(* Logix 5000 project; controller test vendor 1 type 14 code 151 rev 32.13; software revision 32.02; part 4 of 4 *)
(* tags used below, declared in another part *)
   _i : DINT;
   _J : INT;
   _n : DINT;
   _T : DINT;
   _z : DINT;
   AirDown : CAM_PROFILE[1010];
   AirUp : CAM_PROFILE[1010];
   avgCrsDyn : REAL;   // 1 min avg of dynamic respiratory system compliance in ml/cmH2O, from measAvgCalc()
   avgCrsQStat : REAL;   // 1 min avg of quasistatic respiratory system compliance in ml/cmH2O, from measAvgCalc()
   avgFlowImax : REAL;   // 1 min avg of max insp flow in l/min, from measAvgCalc()
   avgMV : REAL;   // 1 min avg of minute ventilation in l/min, from measAvgCalc()
   avgPEEP : REAL;   // 1 min avg of positive end expiratory pressure in cmH2O, from measAvgCalc()
   avgPpeak : REAL;   // 1 min avg of peak insp pressure in cmH2O, from measAvgCalc()
   avgPplat : REAL;   // 1 min avg of plateau insp pressure in cmH2O, from measAvgCalc()
   avgRaw : REAL;   // 1 min avg of airway resistance in cmH2O/l/s, from measAvgCalc()
   avgRR : REAL;   // 1 min avg of respiratory rate in 1/min, from measAvgCalc()
   avgVti : REAL;   // 1 min avg of insp tidal volume in ml, from measAvgCalc()
   BackingTag : MOTION_INSTRUCTION;
   BreathDuration : INT;
   BreathDurationArr : REAL[50];   // 50 length array with seconds for each breath for calculation of minute avgVentStateArr. Calcualted from knowing meas at
   CalcNewData : BOOL;
   CrsDyn : REAL;   // dynamic respiraotry system compliance in ml/cmH2O
   CrsDynArr : REAL[50];   // 50 length array with dynamic respiraotry system compliance in ml/cmH2O, from measCalc()
   CrsQStat : REAL;   // quasistatic respiratory system compliance in ml/cmH2O
   CrsQStatArr : REAL[50];   // 50 length array with quasistatic respiratory system compliance in ml/cmH2O, from measCalc()
   DymmyMaster : AXIS_VIRTUAL;
   DymmySlave : AXIS_VIRTUAL;
   endI : DINT;
   EndPoint : INT;
   Exp : BOOL;
   expEndI : INT;
   expStartI : INT;
   FillLoop : AOI_FillArray_Real2D;
   FlowArrMem : REAL[1000,2];
   FlowImax : REAL;   // max insp flow in l/min
   FlowImaxArr : REAL[50];   // 50 length array with max insp flow in l/min, from measCalc()
   FlowImaxValue : AOI_Max;
   FlowO2Mem : REAL[1000,2];
   i : DINT;
   Insp : BOOL;
   inspPauseStartI : INT;
   inspPauseTimeInMS : REAL;
   inspStartI : INT;
   Mean50 : AOI_Mean50;
   Mode : STRING;
   MV : REAL;   // minute ventilation in l/min
   MVArr : REAL[50];   // 50 length array with minute ventilation in l/min, from measCalc()
   O2Down : CAM_PROFILE[1010];
   O2Up : CAM_PROFILE[1010];
   PEEP : REAL;   // positive end expiratory pressure in cmH2O
   PEEPArr : REAL[50];   // 50 length array with positive end expiratory pressure in cmH2O, from measCalc()
   PEEPi : REAL;
   Ppeak : REAL;   // Ppeak
   PpeakArr : REAL[50];   // 50 length array with Ppeak from measCalc(), used for minAvg
   PpeakMaxValue : AOI_Max;
   Pplat : REAL;   // plateau insp pressure in cmH2O
   PplatArr : REAL[50];   // 50 length array with plateau insp pressure in cmH2O, from measCalc()
   PplatBreathFrac : REAL;
   PplatMean : AOI_Mean2D;
   PressArr : REAL[1000,2];   // 1000 length 2D FIFO array with pressure values and status bits indicating if values have been analysed (1) or not (0) by
   PressArrMem : REAL[1000,2];
   Pressure : REAL;
   Raw : REAL;   // airway resistance in cmH2O/l/s
   RawArr : REAL[50];   // 50 length array with airway resistance in cmH2O/l/s
   Round : AOI_Round;
   RR : REAL;   // respiratory rate in 1/min
   RRArr : REAL[50];   // 50 length array with respiratory rate in 1/min, from measCalc()
   RunModes : STRING[4];
   Samplerate : DINT;   // The rate in Hz that samples is collected
   SetupDone : BOOL;
   SetupState : DINT;
   StartPoint : INT;
   StartPointMean : REAL;
   StartPointValue : REAL;
   state : DINT;
   Time : DINT;
   TimeRate : DINT;
   tipause : INT;
   totTime : INT;
   Vt : INT;   // 200-600 ml
   Vti : REAL;   // insp tidal volume in ml
   VtiArr : REAL[50];   // 50 length array with insp tidal volume in ml, from measCalc()

PROGRAM measCalc   (* main routine Main *)

ROUTINE Main   (* structured text *)
   // from inflow and press alone (may require filtering such as mean/median!)
   // Only check indices with FlowArr[0,x]=0, meaning not analysed yet
   
   if CalcNewData then;
   
   	inspStartI := 0;
   	expStartI := 0;
   	expEndI := 0;
   
   	for _i := 1 to 999 by 1 do
   
   		if FlowArrMem[_i,1] = 0 then;												// Check if data is read already
   
   			if inspStartI = 0 then;													// If Inspiratory start point not found
   
   				//Start of insp is at shift from flow of zero to flow of >0.
   
   				if FlowArrMem[_i-1,0] = 0 and FlowArrMem[_i,0] > 0 then;			// If start of climing flow, were last point was zero and this point has a value
   					inspStartI := _i ;												// Set Inspiratory start point
   				end_if;
   			end_if;
   
   			if inspStartI > 0 and expStartI = 0 then;								// If Inspiratory start point found but nor the Expiratory point
   
   				//Start of exp is at shift from to flow of >0 to flow of zero.
   
   				if FlowArrMem[_i-1,0] > 0 and FlowArrMem[_i,0] = 0 then;			// If end of climing flow, and start of Pplat + Pplat time
   					if Mode = RunModes[0] then;										// If mode is VC
   						inspPauseStartI := _i;										// Set inspiratory pause start point
   						expStartI := _i + ABS(tipause/(TimeRate/1000));				// Set Expiratory start point
   					else
   						expStartI := _i;											// Set Expiratory start point
   					end_if;
   				end_if;
   			end_if;
   
   			if inspStartI > 0 and expStartI > 0 and expEndI = 0 then;				// If Inspiratory start point found and the Expiratory start point, but not Expiratory end point
   
   				//End of exp is at shift from to flow of zero to flow of >0.
   
   				if FlowArrMem[_i-1,0] = 0 and FlowArrMem[_i,0] > 0 then;			// If flow is zero and detection of new breath
   					expEndI := _i - 1;												// Set Expiratory end point
   				end_if;
   			end_if;
   		end_if;
   	end_for;
   
   	// Check of iligal calculation that would bring the controller in Major fault
   	if inspStartI <1 then;
   		inspStartI :=1 ;
   	end_if;
   
   	if expStartI <1 then;
   		expStartI := inspStartI +1;
   	end_if;
   
   	if expEndI < 1 then;
   		expEndI := expStartI +1;
   	end_if;
   
   	// Set all calculations vaerables for breath
   
   	// Breathduration
   	BreathDuration := ((expEndI-inspStartI+1)/Samplerate);
   	RR := (60/BreathDuration);
   
   	// in area with inflow=0 before insp start --> PEEP
   	PEEP := PressArrMem[inspStartI-1,0];
   
   	// in area with inflow=0 check for increase in press (Exp pause, exp flow=0) --> PEEP+PEEPi
   	// NOTE as exp pause cannot be detected this is not possible at the moment,
   	// but should be done here
   	//PEEP := (PEEP+PEEPi)-PEEP;
   
   	// Ppeak = Max pressure during insp
   	// NOTE: will require filtering, e.g. moving average
   
   	AOI_Max(PpeakMaxValue,PressArrMem, 0, inspStartI, expStartI);
   	Ppeak := PpeakMaxValue.Out_Max;
   
   	// Flowi,max = max flow during insp
   	// NOTE: will require filtering e.g. moving average, should be around same
   	// sample range as Ppeak
   	// in VC this is the constant delived level of insp Flow
   
   	AOI_Max(FlowImaxValue, FlowArrMem, 0,inspStartI, expStartI);
   	FlowImax := FlowImaxValue.Out_Max;
   
   	// Pplat = pressure at period immediately following inFlow=0 where
   	// pressure equilibrates
   	// only available if insp pause was performed
   	// Calculated as mean of last fifth of the pause period
   
   	if inspPauseStartI > 0 then;
   		StartPointValue := (inspPauseTimeInMS/1000) * Samplerate*PplatBreathFrac;
   		AOI_Round(Round, StartPointValue, StartPointMean);
   		StartPoint := expStartI-StartPointMean-1;
   		EndPoint := expStartI-1;
   	AOI_Mean2D(PplatMean, PressArrMem, 0, StartPoint, EndPoint);
   		Pplat := PplatMean.Out_Mean;
   	else
   		Pplat := 0;
   	end_if;
   
   	//Vti = integrate inFlow(insp start to exp start)
   
   	for _J := inspStartI to expStartI by 1 do
   	    Vti := Vti + FlowArrMem[_J,0] * (1/(Samplerate*60));
   	end_for;
   
   	//MV = RR*Vti
   
   	MV := RR*Vti;
   
   	//Raw = (Ppeak-Pplat)/Flowi,max    %NOTE: in cmH2O/l/s (different time
   	//unit than Flowi,max at l/min
   	//only available if insp pause was performed so that we have Pplat
   	//assumes FlowIMax is at PIP
   
   	if inspPauseStartI > 0 then;
   	    Raw := (Ppeak-Pplat)/(FlowImax/60);   //FlowIMax/60 to go from l/min to l/s as Raw is in units of l/s
   	else
   	    Raw := 0;
   	end_if;
   
   	//Crs_dyn = Vt/(Ppeak-PEEP)
   	CrsDyn := Vti/(Ppeak-PEEP);
   
   	//Crs_qstat = Vt/(Pplat-PEEP)
   	if inspPauseStartI > 0 then;
   	    CrsQStat := Vti/(Pplat-PEEP);
   	else
   	    CrsQStat := 0;
   	end_if;
   
   
   	//set second dimension status marker in FlowArr and PressArr to 1 from
   	//inspStartI to expEndI to indicate that this breath has been analysed
   	for _n := inspStartI to expEndI+1 by 1 do
   
   		//FlowArrMem[_n,1] := 1;
   		//PressArrMem[_n,1] := 1;
   
   	end_for;
   
   
   	for _T := 49 to 1 by -1 do
   
   		PpeakArr[_T] := PpeakArr[_T-1];
   		PEEPArr[_T] := PEEPArr[_T-1];
   		FlowImaxArr[_T] := FlowImaxArr[_T-1];
   		PplatArr[_T] := PplatArr[_T-1];
   		RRArr[_T] := RRArr[_T-1];
   		VtiArr[_T] := VtiArr[_T-1];
   		MVArr[_T] := MVArr[_T-1];
   		CrsDynArr[_T] := CrsDynArr[_T-1];
   		CrsQStatArr[_T] := CrsQStatArr[_T-1];
   		RawArr[_T] := RawArr[_T-1];
   		BreathDurationArr[_T] := BreathDurationArr[_T-1];
   
   	end_for;
   
   		PpeakArr[0] := Ppeak;
   		PEEPArr[0] := PEEP;
   		FlowImaxArr[0] := FlowImax;
   		PplatArr[0] := Pplat;
   		RRArr[0] := RR;
   		VtiArr[0] := Vti;
   		MVArr[0] := MV;
   		CrsDynArr[0] := CrsDyn;
   		CrsQStatArr[0] := CrsQStat;
   		RawArr[0] := Raw;
   		BreathDurationArr[0] := BreathDuration;
   
   
   	//in case there is not a minute of measurements available yet, then calculate
   	//from the available entries in array
   	//This could be signaled by setting all values in array as -1 until they
   	//have been used, this is done by initVent
   	//I asume here that if an entry is -1 then it is not available
   
   	for _z := 1 to 49 by 1 do
   	    if BreathDurationArr[_z] = -1 and _z = 1 then;
   	        //(disp('error, no breath by breath measurements available');
   	        _z :=50;										// Break the for loop
   	    end_if;
   	    if _z < 50 then;
   			if BreathDurationArr[_z] = -1 then;
   	        	endI := i-1;
   	        	_z :=50;
   			end_if;
   	    end_if;
   
   		if _z < 49 then;
   	    	totTime := totTime+BreathDurationArr[_z];
   		end_if;
   	    if totTime >= 60 then;
   	        endI := _z;
   	        _z :=50;
   	    end_if;
   	end_for;
   
   
   	// Calculate the average from last minute
   
   	AOI_Mean50(Mean50, PpeakArr, 1, endI);			//1 min avg of peak insp pressure in cmH2O
   	avgPpeak :=Mean50.Out_Mean;						// Output of mean
   	AOI_Mean50(Mean50, PEEPArr, 1, endI);			//1 min avg of positive end expiratory pressure in cmH2O
   	avgPEEP :=Mean50.Out_Mean;						// Output of mean
   	AOI_Mean50(Mean50, FlowImaxArr, 1, endI);		//1 min avg of max insp flow in l/min
   	avgFlowImax :=Mean50.Out_Mean;						// Output of mean
   	AOI_Mean50(Mean50, PplatArr, 1, endI);			//1 min avg of plateau insp pressure in cmH2O
   	avgPplat :=Mean50.Out_Mean;						// Output of mean
   	AOI_Mean50(Mean50, RRArr, 1, endI);				//1 min avg of respiratory rate in 1/min
   	avgRR :=Mean50.Out_Mean;						// Output of mean
   	AOI_Mean50(Mean50, VtiArr, 1, endI);			//1 min avg of insp tidal volume in ml
   	avgVti :=Mean50.Out_Mean;						// Output of mean
   	AOI_Mean50(Mean50, MVArr, 1, endI);				//1 min avg of minute ventilation in l/min
   	avgMV :=Mean50.Out_Mean;						// Output of mean
   	AOI_Mean50(Mean50, CrsDynArr, 1, endI);			//1 min avg of dynamic respiratory system compliance in ml/cmH2O
   	avgCrsDyn :=Mean50.Out_Mean;						// Output of mean
   	AOI_Mean50(Mean50, CrsQStatArr, 1, endI);		//1 min avg of quasistatic respiratory system compliance in ml/cmH2O
   	avgCrsQStat :=Mean50.Out_Mean;						// Output of mean
   	AOI_Mean50(Mean50, RawArr, 1, endI);			//1 min avg of airway resistance in cmH2O/l/s
   	avgRaw :=Mean50.Out_Mean;						// Output of mean
   
   	CalcNewData :=0;
   	AOI_FillArray_Real2D(FillLoop,FlowArrMem,0,2000);			// Clear all raw data
   	AOI_FillArray_Real2D(FillLoop,FlowO2Mem ,0,2000);			// Clear all raw data
   	AOI_FillArray_Real2D(FillLoop,PressArrMem,0,2000);			// Clear all raw data
   
   end_if;
END_ROUTINE
END_PROGRAM

PROGRAM Setup   (* main routine Main *)
VAR
   testbit : DINT := 311;
END_VAR

ROUTINE InitGUI   (* structured text *)
   // Init program of the GUI (HMI panel)
   // Write initial coder here
   
   
   
   
END_ROUTINE

ROUTINE InitISR_RS232   (* structured text *)
   // Init program of the ISR_RS232 AI controller
   // Write initial coder here
   
   
   
END_ROUTINE

ROUTINE InitVariables   (* structured text *)
   // Init program of the Init varables for the program
   // Write initial coder here
   
END_ROUTINE

ROUTINE Main   (* structured text *)
   case SetupState of
   
   	10: JSR(InitVariables,0);			// Jump to Init Variables
   		SetupState := 20;				// Set next state
   
   	20:	JSR(InitGUI,0);					// Jump to Init GUI
   		SetupState := 30;				// Set next state
   
   	30:	JSR(InitISR_RS232);				// Jump to init ISR_RS232
   		SetupDone :=1;					// Set Setup Done
   		SetupState := 99;				// Sequence Done
   
   end_case;
END_ROUTINE
END_PROGRAM

PROGRAM ValveProfile   (* main routine Main *)

ROUTINE Main   (* ladder *)
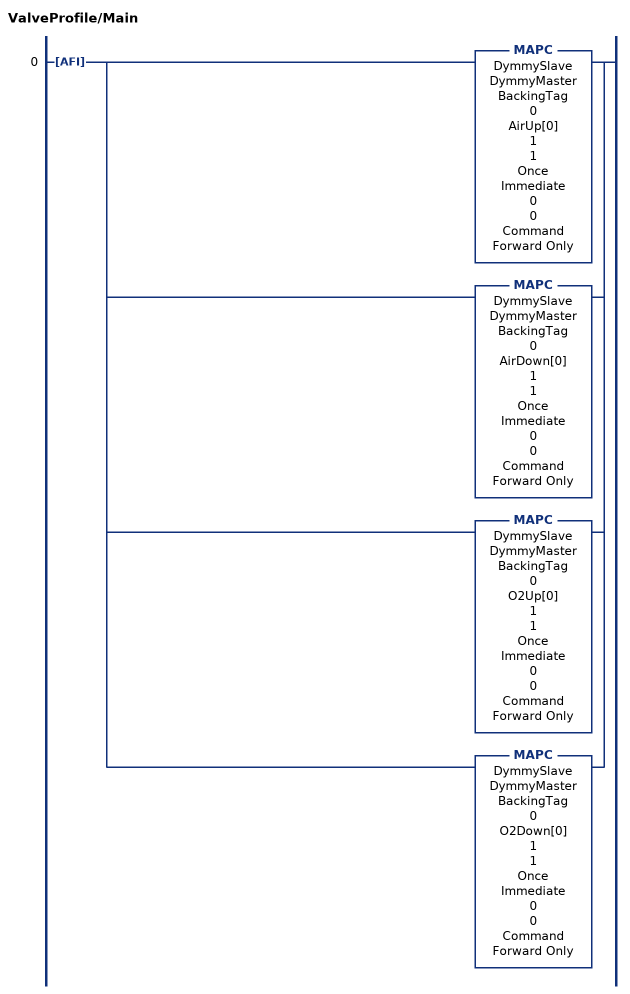
   0: AFI()[MAPC(DymmySlave,DymmyMaster,BackingTag,0,AirUp[0],1,1,Once,Immediate,0,0,Command,Forward Only) ,MAPC(DymmySlave,DymmyMaster,BackingTag,0,AirDown[0],1,1,Once,Immediate,0,0,Command,Forward Only) ,MAPC(DymmySlave,DymmyMaster,BackingTag,0,O2Up[0],1,1,Once,Immediate,0,0,Command,Forward Only) ,MAPC(DymmySlave,DymmyMaster,BackingTag,0,O2Down[0],1,1,Once,Immediate,0,0,Command,Forward Only) ];
END_ROUTINE
END_PROGRAM
